// LS Electric XG5000 project: top2_8_10_검사중1
// PLC LSPLC
// module base 0 slot 0: 입출력 모듈:XBM-DN32H (DC 24V입력/TR 출력, 32점)

PROGRAM NewProgram (task: 스캔 프로그램)

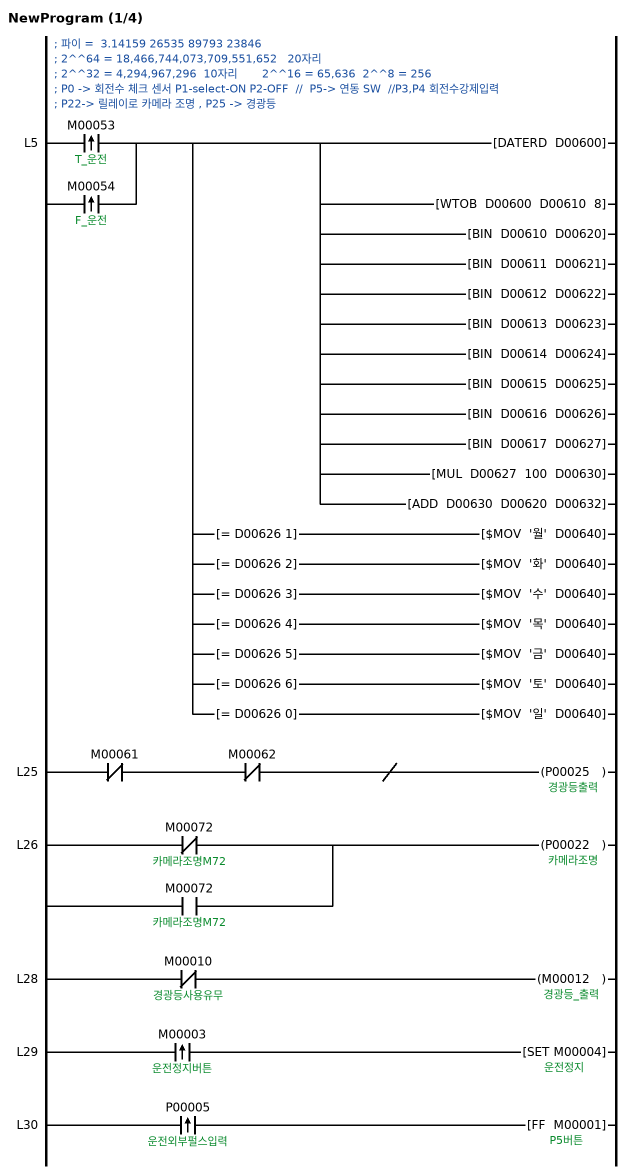
// 파이 =  3.14159 26535 89793 23846
//  2^^64 = 18,466,744,073,709,551,652   20자리
// 2^^32 = 4,294,967,296  10자리       2^^16 = 65,636  2^^8 = 256
//   P0 -> 회전수 체크 센서 P1-select-ON P2-OFF  //  P5-> 연동 SW  //P3,P4 회전수강제입력
//   P22-> 릴레이로 카메라 조명 , P25 -> 경광등
; L5
LOADP     M00053	// T_운전
ORP       M00054	// F_운전
DATERD    D00600
WTOB      D00600 D00610 8
BIN       D00610 D00620
BIN       D00611 D00621
BIN       D00612 D00622
BIN       D00613 D00623
BIN       D00614 D00624
BIN       D00615 D00625
BIN       D00616 D00626
BIN       D00617 D00627
MUL       D00627 100 D00630
ADD       D00630 D00620 D00632
MPUSH
AND=      D00626 1
$MOV      '월' D00640
MLOAD
AND=      D00626 2
$MOV      '화' D00640
MLOAD
AND=      D00626 3
$MOV      '수' D00640
MLOAD
AND=      D00626 4
$MOV      '목' D00640
MLOAD
AND=      D00626 5
$MOV      '금' D00640
MLOAD
AND=      D00626 6
$MOV      '토' D00640
MPOP
AND=      D00626 0
$MOV      '일' D00640
; L25
LOAD NOT  M00061
AND NOT   M00062
NOT
OUT       P00025	// 경광등출력
; L26
LOAD NOT  M00072	// 카메라조명M72
OR        M00072	// 카메라조명M72
OUT       P00022	// 카메라조명
; L28
LOAD NOT  M00010	// 경광등사용유무
OUT       M00012	// 경광등_출력
; L29
LOADP     M00003	// 운전정지버튼
SET       M00004	// 운전정지
; L30
LOADP     P00005	// 운전외부펄스입력
FF        M00001	// P5버튼

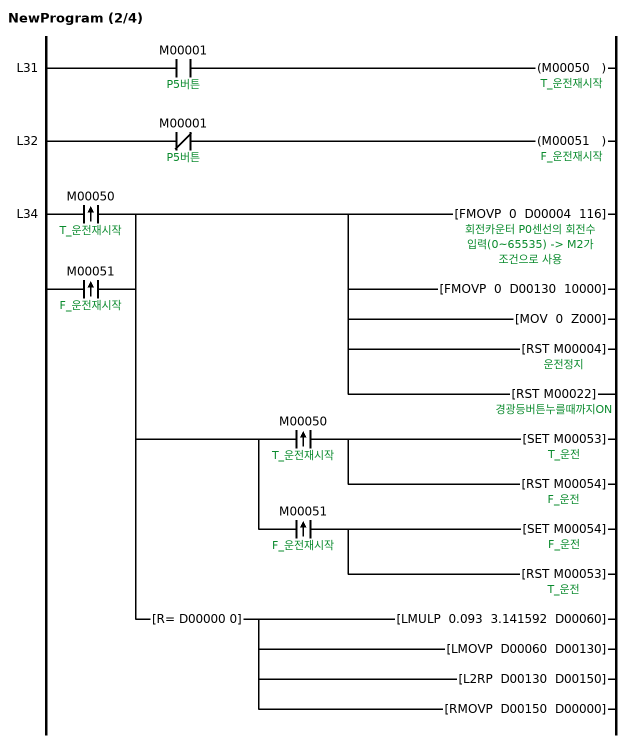
; L31
LOAD      M00001	// P5버튼
OUT       M00050	// T_운전재시작
; L32
LOAD NOT  M00001	// P5버튼
OUT       M00051	// F_운전재시작
; L34
LOADP     M00050	// T_운전재시작
ORP       M00051	// F_운전재시작
FMOVP     0 D00004 116	// 회전카운터 P0센선의 회전수 입력(0~65535) -> M2가 조건으로 사용
FMOVP     0 D00130 10000
MOV       0 Z000
RST       M00004	// 운전정지
RST       M00022	// 경광등버튼누를때까지ON
MPUSH
ANDP      M00050	// T_운전재시작
SET       M00053	// T_운전
RST       M00054	// F_운전
MLOAD
ANDP      M00051	// F_운전재시작
SET       M00054	// F_운전
RST       M00053	// T_운전
MPOP
ANDR=     D00000 0
LMULP     0.093 3.141592 D00060
LMOVP     D00060 D00130
L2RP      D00130 D00150
RMOVP     D00150 D00000

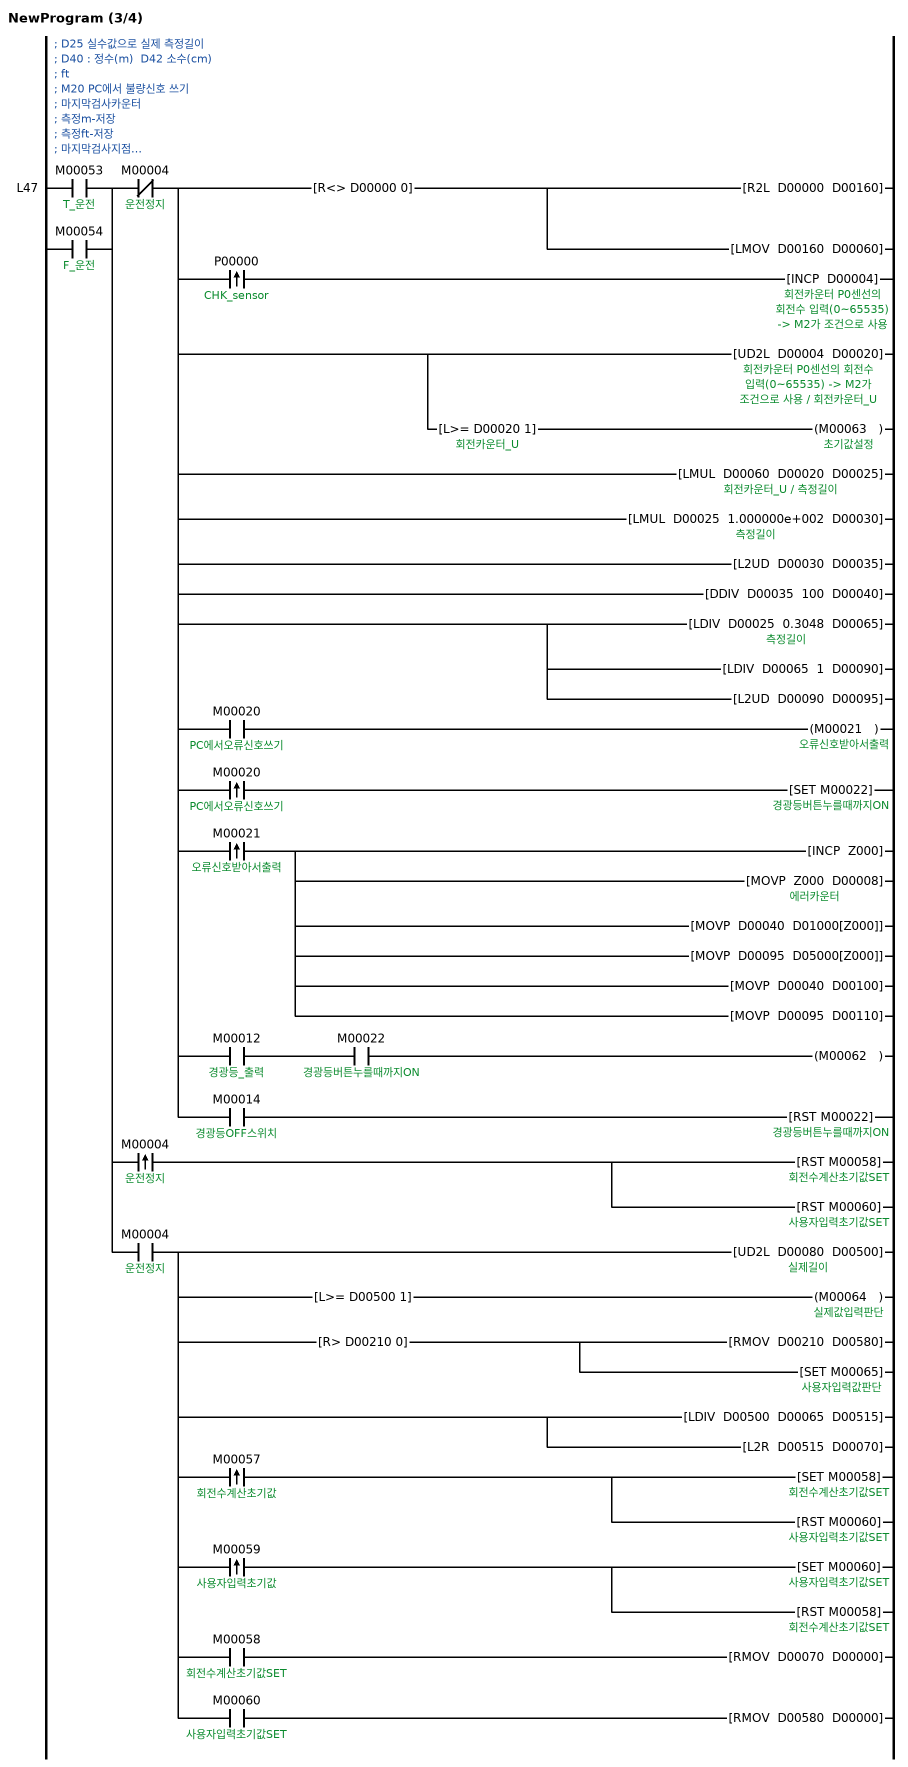
; L47
LOAD      M00053	// T_운전
OR        M00054	// F_운전
MPUSH
AND NOT   M00004	// 운전정지
MPUSH
ANDR<>    D00000 0
R2L       D00000 D00160
LMOV      D00160 D00060
MLOAD
ANDP      P00000	// CHK_sensor
INCP      D00004	// 회전카운터 P0센선의 회전수 입력(0~65535) -> M2가 조건으로 사용
MLOAD
UD2L      D00004 D00020	// 회전카운터 P0센선의 회전수 입력(0~65535) -> M2가 조건으로 사용 / 회전카운터_U
ANDL>=    D00020 1	// 회전카운터_U
OUT       M00063	// 초기값설정
MLOAD
LMUL      D00060 D00020 D00025	// 회전카운터_U / 측정길이
LMUL      D00025 1.000000e+002 D00030	// 측정길이
L2UD      D00030 D00035
DDIV      D00035 100 D00040
LDIV      D00025 0.3048 D00065	// 측정길이
LDIV      D00065 1 D00090
L2UD      D00090 D00095
AND       M00020	// PC에서오류신호쓰기
OUT       M00021	// 오류신호받아서출력
MLOAD
ANDP      M00020	// PC에서오류신호쓰기
SET       M00022	// 경광등버튼누를때까지ON
MLOAD
ANDP      M00021	// 오류신호받아서출력
INCP      Z000
MOVP      Z000 D00008	// 에러카운터
MOVP      D00040 D01000[Z000]
MOVP      D00095 D05000[Z000]
MOVP      D00040 D00100
MOVP      D00095 D00110
MLOAD
AND       M00012	// 경광등_출력
AND       M00022	// 경광등버튼누를때까지ON
OUT       M00062
MPOP
AND       M00014	// 경광등OFF스위치
RST       M00022	// 경광등버튼누를때까지ON
MLOAD
ANDP      M00004	// 운전정지
RST       M00058	// 회전수계산초기값SET
RST       M00060	// 사용자입력초기값SET
MPOP
AND       M00004	// 운전정지
UD2L      D00080 D00500	// 실제길이
MPUSH
ANDL>=    D00500 1
OUT       M00064	// 실제값입력판단
MLOAD
ANDR>     D00210 0
RMOV      D00210 D00580
SET       M00065	// 사용자입력값판단
MLOAD
LDIV      D00500 D00065 D00515
L2R       D00515 D00070
ANDP      M00057	// 회전수계산초기값
SET       M00058	// 회전수계산초기값SET
RST       M00060	// 사용자입력초기값SET
MLOAD
ANDP      M00059	// 사용자입력초기값
SET       M00060	// 사용자입력초기값SET
RST       M00058	// 회전수계산초기값SET
MLOAD
AND       M00058	// 회전수계산초기값SET
RMOV      D00070 D00000
MPOP
AND       M00060	// 사용자입력초기값SET
RMOV      D00580 D00000
// output comment: D25 실수값으로 실제 측정길이
// output comment: D40 : 정수(m)  D42 소수(cm)
// output comment: ft
// output comment: M20 PC에서 불량신호 쓰기
// output comment: 마지막검사카운터
// output comment: 측정m-저장
// output comment: 측정ft-저장
// output comment: 마지막검사지점m
// output comment: ft 검출지점
// output comment: 계산에의한초기값(<-M57
// output comment: 사용자입력초기값(<-M59
// output comment: 실제길이변환
// output comment: 오차율 = 오차/실제값

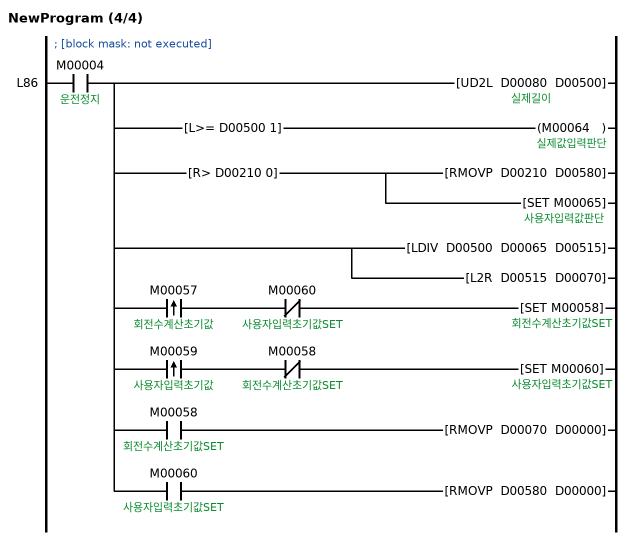
; L86 (block mask: not executed)
LOAD      M00004	// 운전정지
UD2L      D00080 D00500	// 실제길이
MPUSH
ANDL>=    D00500 1
OUT       M00064	// 실제값입력판단
MLOAD
ANDR>     D00210 0
RMOVP     D00210 D00580
SET       M00065	// 사용자입력값판단
MLOAD
LDIV      D00500 D00065 D00515
L2R       D00515 D00070
ANDP      M00057	// 회전수계산초기값
AND NOT   M00060	// 사용자입력초기값SET
SET       M00058	// 회전수계산초기값SET
MLOAD
ANDP      M00059	// 사용자입력초기값
AND NOT   M00058	// 회전수계산초기값SET
SET       M00060	// 사용자입력초기값SET
MLOAD
AND       M00058	// 회전수계산초기값SET
RMOVP     D00070 D00000
MPOP
AND       M00060	// 사용자입력초기값SET
RMOVP     D00580 D00000

VARIABLES AND COMMENTS (devices not used above)
M00008	BIT	CHK_add1 // P0 - 센서입력으로 M8-라이징엣지
M00200	BIT	M0_끄기SW
M00015	BIT	PG_start입력
M00000	BIT	검사시작_PC // 프로그램시작
M00201	BIT	검사종료YES_SW
M00202	BIT	검사종료_NO_SW
M00023	BIT	검사중지로초기화
M00024	BIT	검사중지로초기화입력버튼
M00025	BIT	데이터초기화
D00530	WORD	보정값
D00550	WORD	보정값입력측정길이
D00540	WORD	보정수치
P00020	BIT	스프레이모터
D00505	WORD	오차
D00510	WORD	오차값
D00520	WORD	오차율
D00545	WORD	일회전수치값
P00003	BIT	입력10더하기 // 임시로사용
P00004	BIT	입력200더하기 // 임시로시용
D00120	WORD	제품번호10자리
T0003	BIT/WORD	제품번호입력시간
D00010	WORD	지름X원주율